{attribute 'pack_mode' := '1'}
TYPE ST_GoToCenter EXTENDS ST_MsgToPLC:
STRUCT
    fSpeed		: LREAL;
END_STRUCT
END_TYPE

(* stored: Version 1.1.0.1, ProductVersion 3.1.4022.18
   DUT ST_GoToCenter: Id {d62dccdf-497d-4dd3-aff3-59cf4d317fb3} *)
